///Get the Code from the HRESULT
FUNCTION F_Code : UINT
VAR_INPUT
    hr : HRESULT;
END_VAR
VAR
END_VAR

F_Code := UDINT_TO_UINT(DINT_TO_UDINT(hr) AND 16#0000FFFF);

END_FUNCTION

(* stored: Version 1.1.0.1, ProductVersion 3.1.4019.2
   POU F_Code: Id {8ca8ae97-dd2a-4577-b10c-49cf12ef4b3a}, SpecialFunc None *)
